TYPE PB_UMG604 :
(*Struktur für das Universalmessgerät 604 (Janitza) *)
STRUCT
	ProfilNummer		: BYTE;
	Wirkleistung 		: REAL;
	Blindleistung		: REAL;
	Scheinleistung	: REAL;
	Wirkarbeit		: REAL;
	Blindarbeit		: REAL;
	Scheinarbeit		: REAL;
	DiZaehlstand		: REAL;
	DiZustand		: REAL;
	DiLeistungswert	: REAL;
	NichtBelegt1		: REAL;
	NichtBelegt2		: REAL;
	NichtBelegt3		: REAL;
	NichtBelegt4		: REAL;
	NichtBelegt5		: REAL;
	NichtBelegt6		: REAL;
	NichtBelegt7		: REAL;
	NichtBelegt8		: REAL;
	NichtBelegt9		: REAL;
	NichtBelegt10		: REAL;
	NichtBelegt11		: REAL;
	NichtBelegt12		: REAL;
	NichtBelegt13		: REAL;
	NichtBelegt14		: REAL;
	NichtBelegt15		: REAL;
	NichtBelegt16		: REAL;
	NichtBelegt17		: REAL;
	NichtBelegt18		: REAL;
	NichtBelegt19		: REAL;
	NichtBelegt20		: REAL;
	NichtBelegt21		: REAL;
	NichtBelegt22		: REAL;
END_STRUCT
END_TYPE

(* stored: Version 1.1.0.1, ProductVersion 3.1.4024.9
   DUT PB_UMG604: Id {a66fac40-d058-4339-b429-79a81d56a0fa} *)
